PROGRAM MAIN
VAR
	fbMotor1: fb_motor;
	fbmotor2: fb_motor;
END_VAR


fbMotor1(bStart:= true, bStop:= true, bStatus=> );

END_PROGRAM

(* stored: Version 1.1.0.1, ProductVersion 3.1.4024.11
   POU MAIN: Id {5d7ce718-129a-4ede-b2b8-37034ae92ca0}, SpecialFunc None *)
